//{{V2}}
DATA_BLOCK DB10

AUTHOR:mh
FAMILY:nb
NAME:nb
VERSION:1.0


       STRUCT
         D0:INT
         D1:INT
         D2:INT
         D3:INT
         D4:INT
         D5:INT:=0
         D6:INT:=0
         D7:INT:=0
       END_STRUCT
BEGIN

       D0:=0
       D1:=0
       D2:=0
       D3:=0
       D4:=0
       D5:=0
       D6:=0
       D7:=0
END_DATA_BLOCK
